(* Logix 5000 project; controller EuniceF_ICA18 vendor 1 type 14 code 150 rev 37.11; software revision 37.00 *)

TASK MainTask (continuous, watchdog 500 ms) : MainProgram

MODULES
   Local : vendor 1 type 14 code 150 (Compact 0, rev 37.11)
      Discrete_IO : Embedded (Compact 1, rev 3.1, Output RPI 20 ms)
      Analog_IO : Embedded (Compact 2, rev 1.1, Output RPI 80 ms)
      Counters : Embedded (Compact 3, rev 1.1, Output RPI 20 ms)
END_MODULES

VAR_GLOBAL   (* controller tags *)
   East_Amber : ALIAS FOR Local:1:O.Data.2;
   East_Green : ALIAS FOR Local:1:O.Data.1;
   East_Red : ALIAS FOR Local:1:O.Data.4;
   East_Wapper : ALIAS FOR Local:1:O.Data.15;
   North_Amber : ALIAS FOR Local:1:O.Data.5;
   North_Green : ALIAS FOR Local:1:O.Data.3;
   North_Red : ALIAS FOR Local:1:O.Data.0;
   SEQ : DINT;
   Timer2s : TIMER := (PRE := 2000);
   Timer4s : TIMER := (PRE := 4000);
   Timer6s : TIMER := (PRE := 6000);
END_VAR

PROGRAM MainProgram   (* main routine MainRoutine *)

ROUTINE MainRoutine   (* ladder *)
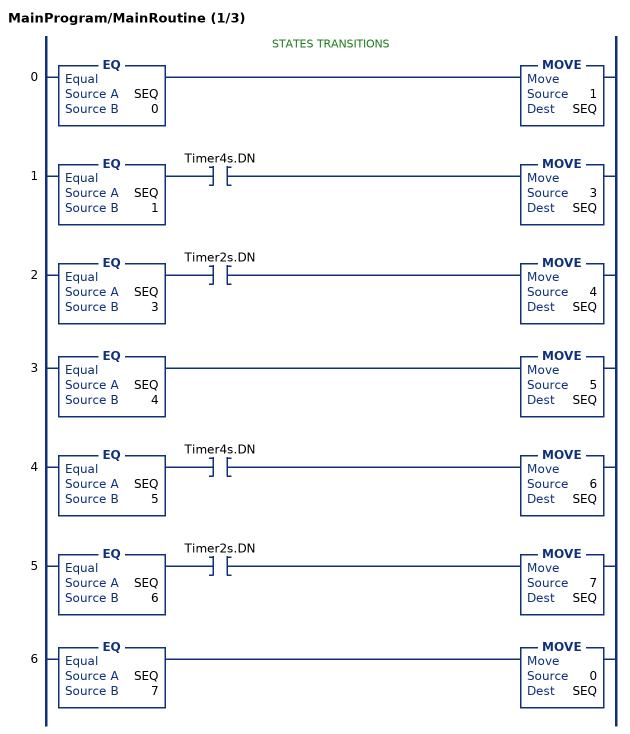
   // STATES TRANSITIONS
   0: EQ(SEQ,0)MOVE(1,SEQ);
   1: EQ(SEQ,1)XIC(Timer4s.DN)MOVE(3,SEQ);
   2: EQ(SEQ,3)XIC(Timer2s.DN)MOVE(4,SEQ);
   3: EQ(SEQ,4)MOVE(5,SEQ);
   4: EQ(SEQ,5)XIC(Timer4s.DN)MOVE(6,SEQ);
   5: EQ(SEQ,6)XIC(Timer2s.DN)MOVE(7,SEQ);
   6: EQ(SEQ,7)MOVE(0,SEQ);
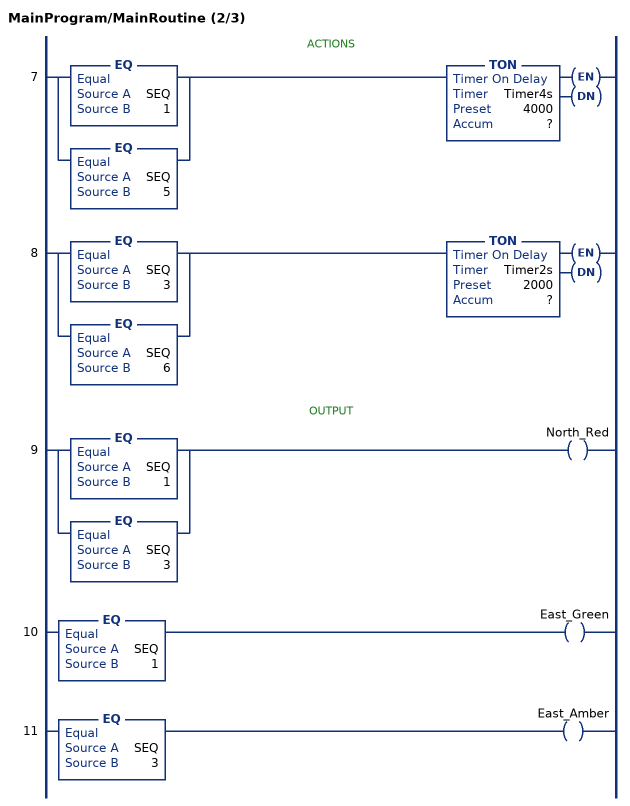
   // ACTIONS
   7: [EQ(SEQ,1) ,EQ(SEQ,5) ]TON(Timer4s,?,?);
   8: [EQ(SEQ,3) ,EQ(SEQ,6) ]TON(Timer2s,?,?);
   // OUTPUT
   9: [EQ(SEQ,1) ,EQ(SEQ,3) ]OTE(North_Red);
   10: EQ(SEQ,1)OTE(East_Green);
   11: EQ(SEQ,3)OTE(East_Amber);
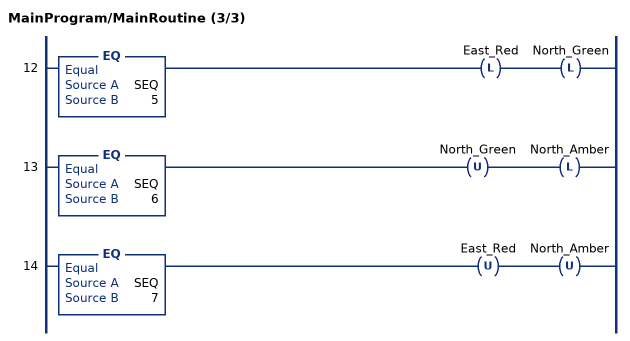
   12: EQ(SEQ,5)OTL(East_Red)OTL(North_Green);
   13: EQ(SEQ,6)OTU(North_Green)OTL(North_Amber);
   14: EQ(SEQ,7)OTU(East_Red)OTU(North_Amber);
END_ROUTINE
END_PROGRAM
